// TwinCAT 3 PLC project FP_OE
// ProgramVersion: 3.1.4023.0
// libraries:
//   Lynus Communicator V2, * (Lynus AG)
//   Tc2_Standard, * (Beckhoff Automation GmbH)
//   Tc2_System, * (Beckhoff Automation GmbH)
//   Tc3_Module, * (Beckhoff Automation GmbH)
// project tree:
//   / Fast.TcTTO, PlcTask.TcTTO, Slow.TcTTO
//   POUs/ MAIN.TcPOU, prgLynusCom.TcPOU, prgLynusVar.TcPOU
// real-time tasks:
//   TASK PlcTask: cycle T#10ms, priority 8, ADS port 350
//   TASK Gerät 1 (OPC UA Virtual)_Task_58: cycle T#40ms, priority 12, ADS port 351
//   TASK Fast: cycle T#5ms, priority 6, ADS port 352
//   TASK Slow: cycle T#20ms, priority 10, ADS port 353
// I/O:
//   DEVICE Gerät 1 (OPC UA Virtual), AmsNetId 172.18.232.244.2.1
// variable links:
//   FP_OE/FP_OE Instance <-> Device 1 (OPC UA Virtual)/Client #1/OPC_HKBKA.OPC_HKBKA.Raumtemperatur_1
//     Slow Inputs/MAIN.rHKBKA_RT1 <-> Inputs/Value
//   FP_OE/FP_OE Instance <-> Device 1 (OPC UA Virtual)/Client #1/OPC_HKBKA.OPC_HKBKA.Raumtemperatur_2
//     Slow Inputs/MAIN.rHKBKA_RT2 <-> Inputs/Value
//   FP_OE/FP_OE Instance <-> Device 1 (OPC UA Virtual)/Client #1/OPC_HKBKA.OPC_HKBKA.Raumtemperatur_3
//     Slow Inputs/MAIN.rHKBKA_RT3 <-> Inputs/Value
//   FP_OE/FP_OE Instance <-> Device 1 (OPC UA Virtual)/Client #1/OPC_HKBKA.OPC_HKBKA.Status_Heizen
//     PlcTask Inputs/MAIN.bStateH <-> Inputs/Value
//   FP_OE/FP_OE Instance <-> Device 1 (OPC UA Virtual)/Client #1/OPC_HKBKA.OPC_HKBKA.Status_Kuehlen
//     PlcTask Inputs/MAIN.bStateC <-> Inputs/Value
//   FP_OE/FP_OE Instance <-> Device 1 (OPC UA Virtual)/Client #1/OPC_HKBKA.OPC_HKBKA.VL_Temp
//     Slow Inputs/MAIN.rHKBKA_FlowT <-> Inputs/Value

CONFIGURATION FP_OE
    RESOURCE PLC ON TwinCAT3
        TASK Fast(INTERVAL := T#5ms, PRIORITY := 6);
        TASK PlcTask(INTERVAL := T#10ms, PRIORITY := 8);
        TASK Slow(INTERVAL := T#20ms, PRIORITY := 10);
        PROGRAM prgLynusVar WITH Fast : prgLynusVar;
        PROGRAM MAIN WITH PlcTask : MAIN;
        PROGRAM prgLynusCom WITH Slow : prgLynusCom;
    END_RESOURCE
END_CONFIGURATION

// ---- POUs/prgLynusVar.TcPOU
PROGRAM prgLynusVar
VAR
	fbVarInfo		: FB_VarInfo;
	fbRW1			: FB_ReadWrite;
	fbRW2			: FB_ReadWrite;
END_VAR

fbVarInfo(
	bReadInfo:= , 
	eTMCFile:= eSelectTMCFile.eDontUseTMCFile, 
	eSavePositionTMCFile:= eSavePositionOnPLC.ePostionC, 
	udiCounterFoundVariables=> , 
	bError=> , 
	bBusy=> , 
	byProgress=> , 
	udiErrorCodeOut=> , 
	eErrorVarInfo_Out=> , 
	sVarWithError=> );
	
fbRW1();
fbRW2();

END_PROGRAM

// ---- POUs/MAIN.TcPOU
PROGRAM MAIN
VAR
	bStateC			AT%I*		: BOOL;
	bStateH			AT%I*		: BOOL;
	byStateH_C					: BYTE;				//{#lynus.ag#()}
	byErrorWarning				: BYTE;				//{#lynus.ag#()}
	byReady						: BYTE;				//{#lynus.ag#()}
	byHB						: BYTE;				//{#lynus.ag#()}
	rHKBKA_RT1	 	AT%I*		: LREAL;			//{#lynus.ag#()}
	rHKBKA_RT2	 	AT%I*		: LREAL;			//{#lynus.ag#()}
	rHKBKA_RT3	 	AT%I*		: LREAL;			//{#lynus.ag#()}
	rHKBKA_FlowT	AT%I*		: LREAL;			//{#lynus.ag#()}
	rNewFlowTemp				: LREAL;			//{#lynus.ag#()}
END_VAR

//State for Heatin gor Cooling
byStateH_C := 0;
	IF bStateC THEN byStateH_C := 2; END_IF
		IF bStateH THEN byStateH_C := 1; END_IF

END_PROGRAM

// ---- POUs/prgLynusCom.TcPOU
PROGRAM prgLynusCom
VAR
	fbCom		: FB_MqttCommunicator;
END_VAR

fbCom(
	bConnect:= TRUE, 
	sUserName:= 'd375c314-cf90-4481-bc8d-a16e93699f17', 
	sUserPassword:= 'd3beadd8-93b3-438b-9d07-f52adf328c7d', 
	eSavePositionCertificate:= eSavePositionOnPLC.ePostionC, 
	bConnected=> , 
	bError=> , 
	hrErrorCode=> , 
	eConnectionState=> , 
	eErrorMessage_Out=> );

END_PROGRAM
